Fanuc KAREL source: KT00635.KL

PROGRAM KT00635
%NOLOCKGROUP
VAR
  Y1: ARRAY[2] OF BYTE
  Y2: ARRAY[2] OF BYTE
  OUT: REAL
BEGIN
  Y1[1] = 2
  Y2[1] = 3
  Y1[1] = 2
  Y2[1] = 3
  OUT = NOT Y1[1]
END KT00635
